{attribute 'linkalways'} 
{attribute 'no_explicit_call' := 'This FB is a CLASS and must be accessed using methods or properties'}
{attribute 'enable_dynamic_creation'}
FUNCTION_BLOCK INTERNAL DefaultMoveVelocityBuilder IMPLEMENTS MoveVelocityBuilder
VAR
	parent_builder : MotionBuilder;
	parameters : REFERENCE TO DefaultBuilderParameters;
	move_absolute_builder : DefaultMoveAbsoluteBuilder(parent_builder := parent_builder, parameters := parameters);
	move_relative_builder : DefaultMoveRelativeBuilder(parent_builder := parent_builder, parameters := parameters);
END_VAR

METHOD PUBLIC Acceleration : MoveVelocityBuilder
VAR_INPUT
	value : LREAL;
END_VAR
parent_builder.Acceleration(value);
Acceleration := THIS^;
END_METHOD

METHOD PUBLIC BufferMode : MoveVelocityBuilder
VAR_INPUT
	mode : MotionBufferMode;
END_VAR
parent_builder.BufferMode(mode);
BufferMode := THIS^;
END_METHOD

METHOD PUBLIC BuildMoveVelocityCommand : MotionCommand
VAR_INPUT
	axis : Axis;
END_VAR
VAR
	command_ptr : POINTER TO MoveVelocityCommand;
	command : MotionCommand;
END_VAR
command_ptr := __NEW(MoveVelocityCommand(
	axis := axis,
	velocity := parameters.velocity,
	acceleration := parameters.acceleration,
	deceleration := parameters.deceleration,
	jerk := parameters.jerk,
	buffer_mode := parameters.buffer_mode
));
BuildMoveVelocityCommand := command_ptr^;
END_METHOD

METHOD PUBLIC Deceleration : MoveVelocityBuilder
VAR_INPUT
	value : LREAL;
END_VAR
parent_builder.Deceleration(value);
Deceleration := THIS^;
END_METHOD

METHOD PUBLIC Distance : MoveRelativeBuilder
VAR_INPUT
	value : LREAL;
END_VAR
parent_builder.Distance(value);
Distance := move_relative_builder;
END_METHOD

//FB_Init is always available implicitly and it is used primarily for initialization.
//The return value is not evaluated. For a specific influence, you can also declare the
//methods explicitly and provide additional code there with the standard initialization
//code. You can evaluate the return value.
METHOD FB_Init: BOOL
VAR_INPUT
    bInitRetains : BOOL; // TRUE: the retain variables are initialized (reset warm / reset cold)
    bInCopyCode : BOOL;  // TRUE: the instance will be copied to the copy code afterward (online change)
	parent_builder : MotionBuilder;
	parameters : REFERENCE TO DefaultBuilderParameters;
END_VAR
THIS^.parent_builder := parent_builder;
THIS^.parameters REF= parameters;
END_METHOD

METHOD PUBLIC Jerk : MoveVelocityBuilder
VAR_INPUT
	value : LREAL;
END_VAR
parent_builder.Jerk(value);
Jerk := THIS^;
END_METHOD

METHOD PUBLIC Position : MoveAbsoluteBuilder
VAR_INPUT
	value : LREAL;
END_VAR
parent_builder.Position(value);
Position := move_absolute_builder;
END_METHOD

METHOD PUBLIC Reset : MoveVelocityBuilder
parent_builder.Reset();
Reset := THIS^;
END_METHOD

METHOD PUBLIC Velocity : MoveVelocityBuilder
VAR_INPUT
	value : LREAL;
END_VAR
parent_builder.Velocity(value);
Velocity := THIS^;
END_METHOD

END_FUNCTION_BLOCK

(* stored: Version 1.1.0.1
   POU DefaultMoveVelocityBuilder: Id {f9842e00-9f13-4dfb-a4fc-1334fd6a45e4}, SpecialFunc None
   Folder Builders: Id {940e7cc8-8a23-4c94-a6aa-ede706520837}
   Folder Constructor: Id {4da8724e-7b13-4591-8b4d-909a298b2caf}
   Folder PropertySetters: Id {eee355ac-afe4-459f-b5f1-a5b199356104}
   Method Acceleration: Id {1b535e18-fab7-4b4d-9048-2e52b44254d5}
   Method BufferMode: Id {1b710cb4-492b-44ac-9bbb-1b625ea1502b}
   Method BuildMoveVelocityCommand: Id {9f3fc142-58fe-08d5-0e8b-502b0083054d}
   Method Deceleration: Id {b8d737be-440a-46ad-aeba-ef6322405832}
   Method Distance: Id {14c1fafb-9242-4670-adee-c4afa17cb820}
   Method FB_Init: Id {c1cd9a84-cc97-4e04-8ded-f872444c78e4}
   Method Jerk: Id {b1b29764-2a12-40e1-88be-3c5a91bcd0cc}
   Method Position: Id {7b33485a-77f8-4919-ba24-8faf5ef3008f}
   Method Reset: Id {b3b36beb-20c2-40b4-a5ef-d61d13b6f149}
   Method Velocity: Id {96c770c8-74af-4b0c-a2e2-e61fe7a41024} *)
